{attribute 'reflection'}
FUNCTION_BLOCK PUBLIC FB_DevHDAnalogInput EXTENDS FB_DevBase
VAR_INPUT
	bCmdSimulate	: BOOL 	:= FALSE ;// Simulate sensor Input 
	fSimValue		: DINT	:= 0 ;// Simulated sensor state
END_VAR
VAR_OUTPUT
	fValue	: LREAL := 0 ; // Analog input value (LREAL)
END_VAR
VAR
	nLimitMin			: DINT := IBF_Utilities.GVL_FixedValues.nDINTMINVALUE	; // Initial value is set to integer minimum value for use with normal def analog inputs 
	nLimitMax 			: DINT := IBF_Utilities.GVL_FixedValues.nDINTMAXVALUE 	; // Initial value is set to integer minimum value for use with high def analog inputs
	inHwInput 	AT%I* 	: DINT ; // Hardware connection
	inStatus	AT%I* 	: BYTE; // input card hardware status
END_VAR

// Set device type
eDevType := E_Devices.AnalogSensor ;

// Call base function
SUPER^();

// Check Hardware connection
CheckHardware();

// set feedback
ExecSetFeedback();

METHOD CheckHardware : BOOL
VAR_INPUT
END_VAR
// Check for hardware faults
IF inStatus.0 THEN // signal under range
	stFault.Active			:= TRUE 							;
	stFault.Description		:= 'Signal under Range';
	stFault.FaultType		:= E_FaultTypes.CF 					;
	bErrorActive			:= TRUE 							;
END_IF

IF inStatus.1 THEN // signal over range
	stFault.Active			:= TRUE 							;
	stFault.Description		:= 'Signal over Range';
	stFault.FaultType		:= E_FaultTypes.CF 					;
	bErrorActive			:= TRUE 							;
END_IF

IF inStatus.6 THEN // general Error bit
	stFault.Active			:= TRUE 							;
	stFault.Description		:= 'Hardware general Error';
	stFault.FaultType		:= E_FaultTypes.FF 					;
	bErrorActive			:= TRUE 							;
END_IF
END_METHOD

METHOD ExecSetFeedback : BOOL
VAR_INPUT
END_VAR
IF bCmdSimulate THEN 
	fValue := fSimValue ;
ELSE
	fValue := DINT_TO_LREAL(inHwInput);
END_IF

ExecSetFeedback := TRUE;
END_METHOD

METHOD PUBLIC Init : BOOL
VAR_INPUT
	// Location data for messages  
	nId			: UINT ; // Identification number of object
	nParentId	: UDINT ; // Id of higher level If aplicable (0 = no parent)
END_VAR
// ====== Set init to true =====
	bInitOk	:= TRUE ; 

// ====== Calculate device id =====
	bInitOk :=	ExecIdentifyDevice(nId,nParentId, E_ComponentTypes.AnInput) AND bInitOk;

// ====== Set feedback =====
	Init := bInitOk ;
END_METHOD

END_FUNCTION_BLOCK

(* stored: Version 1.1.0.1, ProductVersion 3.1.4024.11
   POU FB_DevHDAnalogInput: Id {17595e23-620c-00d9-1a3c-cd0af05163c6}, SpecialFunc None
   Method CheckHardware: Id {de66372f-1f59-079d-284f-b942f3a56b98}
   Method ExecSetFeedback: Id {e186a48a-464f-020c-23e9-d266b6ce2852}
   Method Init: Id {89115260-2041-0458-044d-7546366459ec} *)
